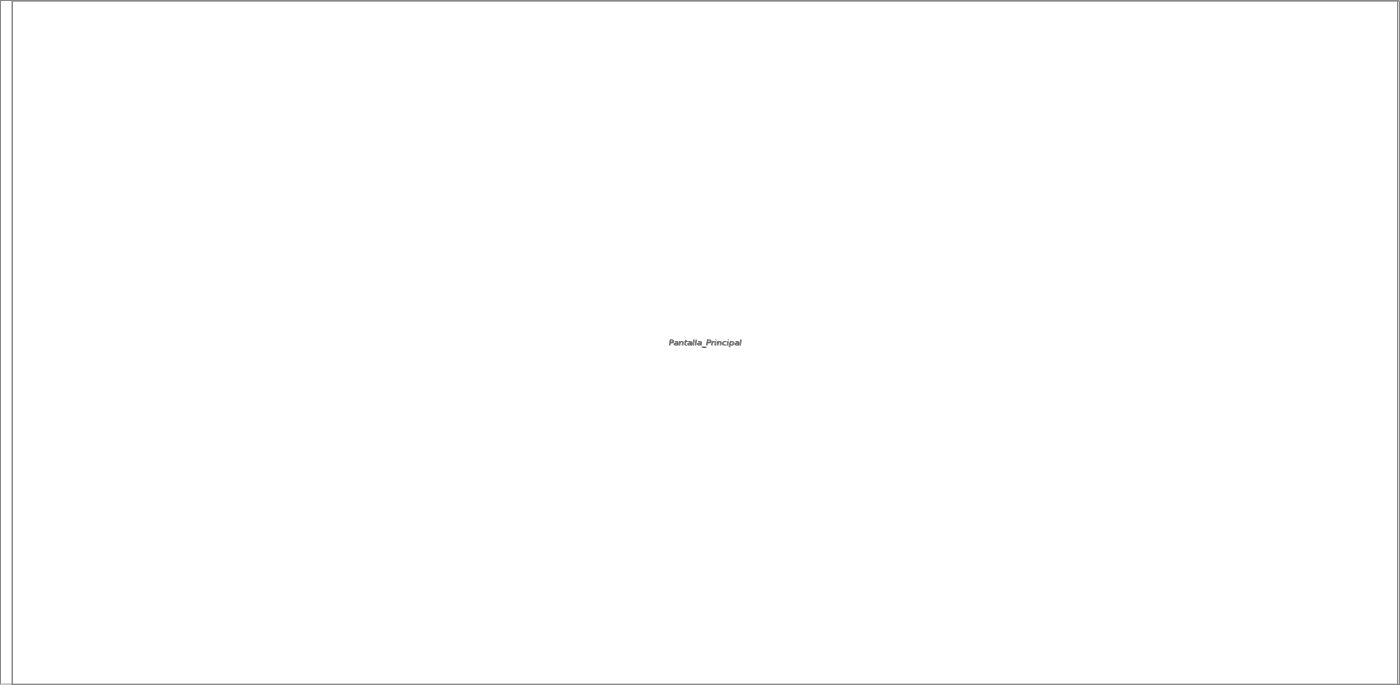
VISUALIZATION HMI  // 1709x837
    TabControl (15,0 1691x837), invisible if: NOT GVL.Manual
        shows Pantalla_Principal()
        shows Entrada_Manual()
        shows Linea_Produccion_Azul_1()
        shows Linea_Produccion_Azul_2()
        shows Linea_Almacen_Manual()
        shows Almacen_Manual()
        shows Senales()
        [0]: TabTitle=Global
        [1]: TabTitle=Entrada
        [2]: TabTitle=Comienzo Producción Azul
        [3]: TabTitle=Final Producción Azul
        [4]: TabTitle=Línea Almacén
        [5]: TabTitle=Entrada Almacen
        [6]: TabTitle=Señales
    TabControl (14,1 1695x836), invisible if: GVL.Manual
        shows Pantalla_Principal()
        shows Entrada_Manual()
        shows Linea_Produccion_Azul_1()
        shows Linea_Produccion_Azul_2()
        shows Linea_Almacen_Manual()
        shows Almacen_Manual()
        shows Senales()
        [0]: TabTitle=Global
        [1]: TabTitle=Entrada
        [2]: TabTitle=Comienzo Linea Azul
        [3]: TabTitle=Final Linea Azul
        [4]: TabTitle=Linea Almacen
        [5]: TabTitle=Entrada Almacen
        [6]: TabTitle=Señales
END_VISUALIZATION

(* stored: Version 1.1.0.1, ProductVersion 3.1.4024.12
   Visu HMI: Id {da646631-6e12-4a4b-8544-82d0c0fdd2af} *)
